Staubli VAL3: trajBuffer.pgx

public program trajBuffer(num x_nElems, num x_nPtsPopped)
begin

  // Do nothing
  // See start() program for more details

end
